Staubli VAL3: yes_no_cancel.pgx

public program yes_no_cancel(string x_sMessage (dimensions=1), string& x_sYesNo[] (dimensions=1), bool& x_bResult[] (dimensions=1), bool& x_bCancel[] (dimensions=1))
  local num i
  local string l_sButton[3]
begin
  // INIT
  x_bCancel=false
  l_sButton[0]=x_sYesNo
  l_sButton[1]=x_sYesNo[1]
  l_sButton[2]="Esc"
  // write a yes no cancel question dialog
  call questionDialog(x_sMessage,l_sButton,i)
  // press F8 or enter
  if i==1 or i==0
    x_bResult=true
  else
    // press escape or F6
    if i==-1 or i==3
      x_bCancel=true
    endIf
    // press F7-no
    x_bResult=false
  endIf
end
